// TIA Portal V17 export
BLOCK "FC_Latch"   // ObjectSW11, LAD
BEGIN

REGION Network 1: sr rs boxes
END_REGION
END_BLOCK
